FUNCTION TryConvert_UINT_TO_DINT : BOOL
VAR_INPUT
	in : UINT;
	out : REFERENCE TO DINT;
END_VAR

out := UINT_TO_DINT(in);
TryConvert_UINT_TO_DINT := TRUE;

END_FUNCTION

(* stored: Version 1.1.0.1, ProductVersion 3.1.4024.12
   POU TryConvert_UINT_TO_DINT: Id {b889ea89-3a4a-4a30-bd37-8fcc9d4d2c3c}, SpecialFunc None *)
